PROGRAM Sequence
VAR
	ePulseState : E_PulseState;
	//eCommand	: E_Command;
	i : INT := 1; //1-8 chargers
	j : INT := 1; //section 1-3
	k : INT := 1; //section 1- 4 
	
	//ChrgRlyHVON_TON : TON;
	//ChrgRlyHVON_PT 	: TIME := T#250MS;
	//ChrgRlyHVON_ET 	: TIME;
END_VAR


//charge command from screen room
IF MCP_IO.CloseAllChargeRlyCommand = TRUE THEN
	//CLOSE ALL CHARGE RELAYS	
	FOR j := 1 TO 3 BY 1 DO
		LCP.Section[j].Peak.CloseChargeRelay1 := TRUE;
		LCP.Section[j].Peak.CloseChargeRelay2 := TRUE;
		LCP.Section[j].Sust.CloseChargeRelay1 := TRUE;
		LCP.Section[j].Sust.CloseChargeRelay2 := TRUE;
	END_FOR;
	LCP.Section[4].Form.CloseChargeRelay1 := TRUE;
	LCP.Section[4].Form.CloseChargeRelay2 := TRUE;
							
	LCP.Section[4].Form.ClosePreFormChargeRly := TRUE;
	LCP.Section[4].Form.CloseFormTrigChargeRly := TRUE;
	LCP.Section[4].Form.ClosePreFormTrigChargeRly := TRUE;
				
ELSE
	//OPEN ALL CHARGE RELAYS	
	FOR j := 1 TO 3 BY 1 DO
		LCP.Section[j].Peak.CloseChargeRelay1 := FALSE;
		LCP.Section[j].Peak.CloseChargeRelay2 := FALSE;
		LCP.Section[j].Sust.CloseChargeRelay1 := FALSE;
		LCP.Section[j].Sust.CloseChargeRelay2 := FALSE;
	END_FOR;
	LCP.Section[4].Form.CloseChargeRelay1 := FALSE;
	LCP.Section[4].Form.CloseChargeRelay2 := FALSE;
							
	LCP.Section[4].Form.ClosePreFormChargeRly := FALSE;
	LCP.Section[4].Form.CloseFormTrigChargeRly := FALSE;
	LCP.Section[4].Form.ClosePreFormTrigChargeRly := FALSE;
END_IF;

//use this for the slim only  -- it will be replaced with the Permissives block for the next upgrade
(*IF Permissives_DB.AllChargeRelaysClosed = TRUE THEN 
		//system ready to charge LED On
		FOR k := 1 TO 4	BY 1 DO 
			LCP.Section[k].SystemReadyToCharge := TRUE;
		END_FOR;
	ELSE
		//system ready to charge LED On
		FOR k := 1 TO 4	BY 1 DO 
			LCP.Section[k].SystemReadyToCharge := FALSE;
		END_FOR;
END_IF;
*)
//open dump command from screen room
IF MCP_IO.OpenAllDumpRelayCommand = TRUE THEN			
	//Open all dump relays 
	FOR j := 1 TO 3 BY 1 DO						
		LCP.Section[j].Peak.OpenDumpRelay1 := TRUE;
		LCP.Section[j].Peak.OpenDumpRelay2 := TRUE;
		LCP.Section[j].Sust.OpenDumpRelay1 := TRUE;
		LCP.Section[j].Sust.OpenDumpRelay2 := TRUE;
							
		LCP.Section[4].Form.OpenDumpRelay1 := TRUE;
		LCP.Section[4].Form.OpenDumpRelay2 := TRUE;
		LCP.Section[4].Form.OpenPreFormDumpRly	:= TRUE;
		LCP.Section[4].Form.OpenFormTrigDumpRly1 := TRUE;
		LCP.Section[4].Form.OpenPreFormTrigDumpRly1 := TRUE;
	END_FOR;
ELSE
	//Close all dump relays 
	FOR j := 1 TO 3 BY 1 DO						
		LCP.Section[j].Peak.OpenDumpRelay1 := FALSE;
		LCP.Section[j].Peak.OpenDumpRelay2 := FALSE;
		LCP.Section[j].Sust.OpenDumpRelay1 := FALSE;
		LCP.Section[j].Sust.OpenDumpRelay2 := FALSE;
							
		LCP.Section[4].Form.OpenDumpRelay1 := FALSE;
		LCP.Section[4].Form.OpenDumpRelay2 := FALSE;
		LCP.Section[4].Form.OpenPreFormDumpRly	:= FALSE;
		LCP.Section[4].Form.OpenFormTrigDumpRly1 := FALSE;
		LCP.Section[4].Form.OpenPreFormTrigDumpRly1 := FALSE;
	END_FOR;
END_IF;

//mapping to the MCP for slim configuration
MCP_IO.AllChargeRelaysClose := Permissives_DB.AllChargeRelaysClosed;
MCP_IO.AllDumpRelaysOpen := Permissives_DB.AllDumpRelaysOpen;


//no sequencing needed************************************************************************************************
(*
//IF BOTH Close charge and open dump signals are off go to idle.
IF MCP_IO.CloseAllChargeRlyCommand = FALSE AND MCP_IO.OpenAllDumpRelayCommand = FALSE THEN
	ePulseState := E_PulseState.SAFE;
END_IF;




//screen room asks to go to close all charge relays when the dump relays are closed ** this should never happen
IF MCP_IO.CloseAllChargeRlyCommand = TRUE AND MCP_IO.OpenAllDumpRelayCommand = FALSE THEN
	ePulseState := E_PulseState.TRIPPED;
END_IF;

//screen room asks to go to open all charge relays when the dump relays are open ** this should never happen - floating system
(*
IF MCP_IO.CloseAllChargeRlyCommand = FALSE AND MCP_IO.OpenAllDumpRelayCommand = TRUE THEN
	//both charge and dump open - floating
END_IF;
*)


CASE ePulseState OF 
	//SAFE / IDLE state
	E_PulseState.SAFE:
							
						//IF no fault and charge permissions and charge relay go to charge mode
						IF MCP_IO.CloseAllChargeRlyCommand = TRUE AND MCP_IO.OpenAllDumpRelayCommand = TRUE THEN
							ePulseState := E_PulseState.CHARGING;
						END_IF;

	//CHARGING STATE
	E_PulseState.CHARGING:
							//turn on charger inhibit
							FOR i := 1 TO 8 BY 1 DO
								MCP_IO.Charger[i].inhibit := TRUE;
							END_FOR;
							
							//Open all dump relays first
							LCP.Bank[j].Peak.OpenDumpRelay1 := TRUE;
							LCP.Bank[j].Peak.OpenDumpRelay2 := TRUE;
							LCP.Bank[j].Sust.OpenDumpRelay1 := TRUE;
							LCP.Bank[j].Sust.OpenDumpRelay2 := TRUE;
							
							LCP.Bank[4].Form.OpenDumpRelay1 := TRUE;
							LCP.Bank[4].Form.OpenDumpRelay2 := TRUE;
							LCP.Bank[4].OpenPreFormDumpRly	:= TRUE;
							LCP.Bank[4].OpenFormTrigDumpRly1 := TRUE;
							LCP.Bank[4].OpenPreFormTrigDumpRly1 := TRUE;
							
							
							
							
							
							//CLOSE ALL CHARGE RELAYS	
							FOR j := 1 TO 3 BY 1 DO
								LCP.Bank[j].Peak.CloseChargeRelay1 := TRUE;
								LCP.Bank[j].Peak.CloseChargeRelay2 := TRUE;
								LCP.Bank[j].Sust.CloseChargeRelay1 := TRUE;
								LCP.Bank[j].Sust.CloseChargeRelay2 := TRUE;
							END_FOR;
							LCP.Bank[4].Form.CloseChargeRelay1 := TRUE;
							LCP.Bank[4].Form.CloseChargeRelay2 := TRUE;
							
							LCP.Bank[4].ClosePreFormChargeRly := TRUE;
							LCP.Bank[4].CloseFormTrigChargeRly := TRUE;
							LCP.Bank[4].ClosePreFormTrigChargeRly := TRUE;
				
							IF MCP_IO.AllChargeRelaysClose = TRUE THEN
								//system ready to charge LED On
								FOR k := 1 TO 4	BY 1 DO 
									LCP.Bank[k].SystemReadyToCharge := TRUE;
								END_FOR;							
						
								//enable all HV ON output and remove inhitbit signal
								FOR i := 1 TO 8 BY 1 DO 
									MCP_IO.Charger[i].HV_ON := TRUE;
									MCP_IO.Charger[i].inhibit := TRUE;
								END_FOR;
								
							ELSE 
								//system ready to charge LED Off
								FOR k := 1 TO 4	BY 1 DO 
									LCP.Bank[k].SystemReadyToCharge := FALSE;
								END_FOR;
									
								FOR i := 1 TO 8 BY 1 DO 
									MCP_IO.Charger[i].HV_ON := FALSE;
								END_FOR;
							END_IF;
							
							//if screen room ask to go the dump
							IF MCP_IO.OpenAllDumpRelayCommand = FALSE AND MCP_IO.CloseAllChargeRlyCommand = FALSE THEN
								ePulseState := E_PulseState.DUMPING;
							END_IF;
	
	//DUMP STATE
	E_PulseState.DUMPING:
							//turn off charger HV ON and Inhibit signals
							FOR i := 1 TO 8 BY 1 DO 
								MCP_IO.Charger[i].HV_ON := FALSE;
								MCP_IO.Charger[i].inhibit := FALSE;
							END_FOR; 
							
							IF MCP_IO.AllChargerHVisON = FALSE THEN
								//Open ALL CHARGE RELAYS	
								FOR j := 1 TO 3 BY 1 DO
									LCP.Bank[j].Peak.CloseChargeRelay1 := FALSE;
									LCP.Bank[j].Peak.CloseChargeRelay2 := FALSE;
									LCP.Bank[j].Sust.CloseChargeRelay1 := FALSE;
									LCP.Bank[j].Sust.CloseChargeRelay2 := FALSE;
								END_FOR;
								LCP.Bank[4].Form.CloseChargeRelay1 := FALSE;
								LCP.Bank[4].Form.CloseChargeRelay2 := FALSE;
							
								LCP.Bank[4].ClosePreFormChargeRly := FALSE;
								LCP.Bank[4].CloseFormTrigChargeRly := FALSE;
								LCP.Bank[4].ClosePreFormTrigChargeRly := FALSE;
							END_IF;
							
							FOR j := 1 TO 3 BY 1 DO 
								LCP.Bank[j].Peak.OpenDumpRelay1 := FALSE;
								LCP.Bank[j].Peak.OpenDumpRelay2 := TRUE;
								LCP.Bank[j].Peak.OpenDumpRelay2 := TRUE;
							END_FOR;
						
	
	//TRIPPED STATE
	E_PulseState.TRIPPED:
							//DO SOMETHING
	
	
	
	
	
END_CASE;
*)
//**********************************************************************************	




IF i > 8 THEN
	i := 1;
END_IF;

IF j > 3 THEN
	j := 1;
END_IF;

IF k > 4 THEN
	k := 1;
END_IF;

END_PROGRAM

(* stored: Version 1.1.0.1, ProductVersion 3.1.4024.11
   POU Sequence: Id {663eae43-1137-476a-a586-15717a445f9e}, SpecialFunc None *)
